(* IEC 61131-3 sources: RL_MAR/experiments/comparison/llm4plc/results/gpt-4o_20260507_114630/20260507_115626, 1 file *)

(* ---- generated_code_iteration_0.st ---- *)
plaintext
START_ST

FUNCTION_BLOCK SmartIrrigationSystem
VAR_INPUT
    SoilMoistureSensor1 : REAL; // Input from the first soil moisture sensor
    SoilMoistureSensor2 : REAL; // Input from the second soil moisture sensor
    WeatherForecast : INT;     // Input for the weather forecast (0: Sunny, 1: Rainy, 2: Cloudy)
END_VAR

VAR_OUTPUT
    WaterPump : BOOL;          // Output to control the water pump
END_VAR

VAR
    state : INT := 0;                  // The current state of the system
    prevState : INT := 0;             // The previous state of the system
    SoilMoistureThreshold : REAL := 30.0; // The threshold for soil moisture
END_VAR

// Main logic for the finite state machine
IF state = 0 THEN
    // STATE 0: IDLE
    WaterPump := FALSE; // Ensure the pump is off
    prevState := state; // Store the previous state
    state := 1;         // Transition to STATE 1 to check conditions

ELSIF state = 1 THEN
    // STATE 1: CHECK CONDITIONS
    WaterPump := FALSE; // Ensure the pump remains off while checking conditions

    IF (WeatherForecast = 0) AND
       ((SoilMoistureSensor1 < SoilMoistureThreshold) OR (SoilMoistureSensor2 < SoilMoistureThreshold)) THEN
        // Transition to STATE 2 to activate the pump
        prevState := state;
        state := 2;

    ELSIF WeatherForecast = 1 THEN
        // Transition to STATE 3 to deactivate the pump
        prevState := state;
        state := 3;

    ELSIF (WeatherForecast <> 0) AND (WeatherForecast <> 1) AND
          (SoilMoistureSensor1 >= SoilMoistureThreshold) AND (SoilMoistureSensor2 >= SoilMoistureThreshold) THEN
        // Transition back to STATE 0 (IDLE)
        prevState := state;
        state := 0;
    END_IF

ELSIF state = 2 THEN
    // STATE 2: ACTIVATE PUMP
    WaterPump := TRUE; // Turn the pump ON
    prevState := state; // Store the previous state
    state := 1;         // Transition back to STATE 1 to re-evaluate conditions

ELSIF state = 3 THEN
    // STATE 3: DEACTIVATE PUMP
    WaterPump := FALSE; // Turn the pump OFF
    prevState := state; // Store the previous state
    state := 1;         // Transition back to STATE 1 to re-evaluate conditions

END_IF

END_FUNCTION_BLOCK

END_ST
